{attribute addProperty BoxType "EK1100-0000-0018"}
{attribute addProperty Id "Beckhoff_EK12xxEK1122Beckhoff_EK12xxEK1122_E9998301162"}
{attribute addProperty CRC "654130762"}
{attribute addProperty SizeInBites "16"}
{attribute addProperty SizeInBytes "2"}
TYPE Beckhoff_EK12xx_26FD3E4A EXTENDS EK1100_179A0949 :
STRUCT
	{attribute addProperty Name "Beckhoff_EK12xxEK1122"}
	Beckhoff_EK12xxEK1122 : Beckhoff_EK12xxEK1122_E9998301;
END_STRUCT
END_TYPE

(* stored: Version 1.2.0.0, ProductVersion 3.1.4024.9
   DUT Beckhoff_EK12xx_26FD3E4A: Id {23003a4f-3464-4a56-aeb9-83c0031f9b27} *)
